{attribute 'qualified_only'}
//{attribute 'strict'}
TYPE Surface :
(
	TOP,
	LEFT,
	RIGHT,
	BOTTOM,
	
	TOP_LEFT,
	TOP_RIGHT,
	BOTTOM_LEFT,
	BOTTOM_RIGHT,
	
	size
);
END_TYPE

(* stored: Version 1.1.0.1, ProductVersion 3.1.4024.11
   DUT Surface: Id {2f7ba695-da26-452c-a259-08ff60ae050e} *)
